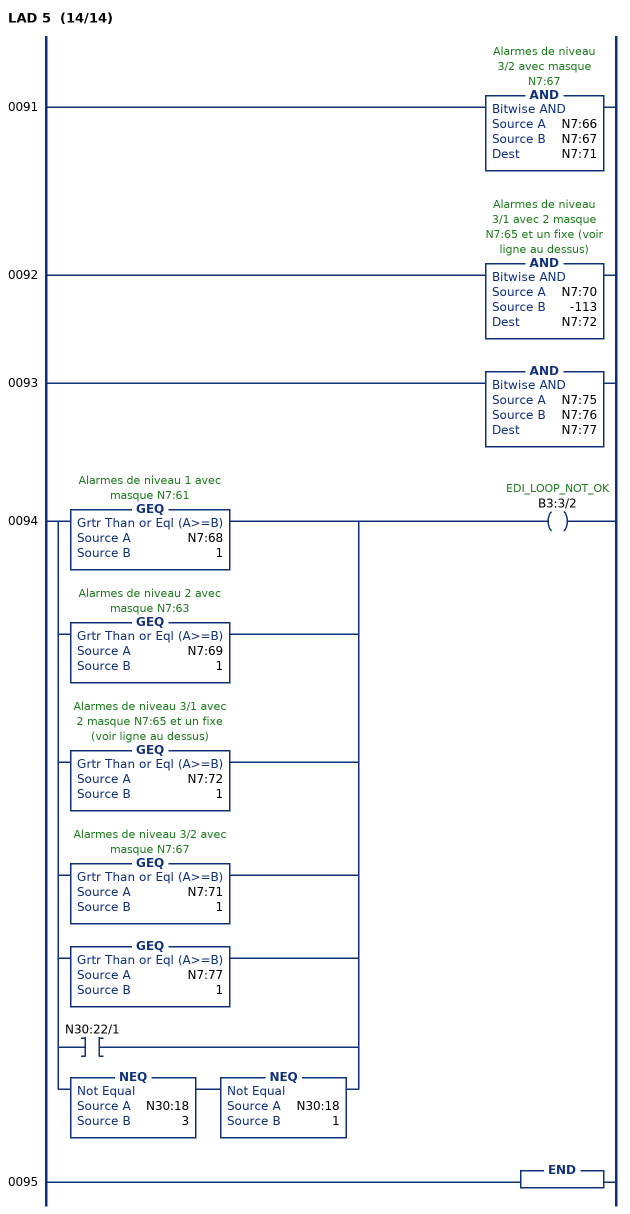
% Rung: 91 %
SOR AND N7:66 N7:67 N7:71 EOR
%   N7:71  "Alarmes de niveau 3/2 avec masque N7:67" %
% Rung: 92 %
SOR AND N7:70 -113 N7:72 EOR
%   N7:70  "Alarmes de niveau 3/1 avec masque N7:65" %
%   N7:72  "Alarmes de niveau 3/1 avec 2 masque N7:65 et un fixe (voir ligne au dessus)" %
% Rung: 93 %
SOR AND N7:75 N7:76 N7:77 EOR
% Rung: 94 %
SOR BST GEQ N7:68 1 NXB GEQ N7:69 1 NXB GEQ N7:72 1 NXB GEQ N7:71 1 NXB GEQ N7:77 1 NXB XIC N30:22/1 NXB NEQ N30:18 3 NEQ N30:18 1 BND OTE B3:3/2 EOR
%   N7:68  "Alarmes de niveau 1 avec masque N7:61" %
%   N7:69  "Alarmes de niveau 2 avec masque N7:63" %
%   N7:72  "Alarmes de niveau 3/1 avec 2 masque N7:65 et un fixe (voir ligne au dessus)" %
%   N7:71  "Alarmes de niveau 3/2 avec masque N7:67" %
%   B3:3/2  EDI_LOOP_NOT_OK %
% Rung: 95 %
SOR END EOR

LADDER 6
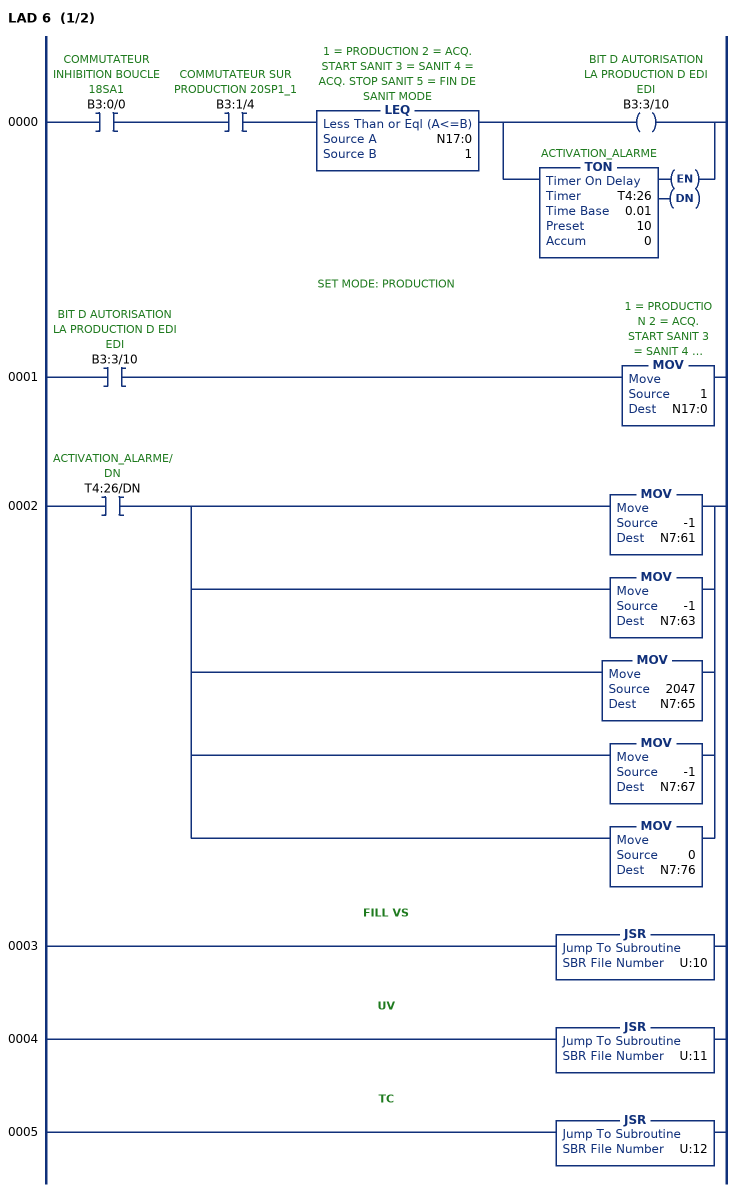
% Rung: 0 %
SOR XIC B3:0/0 XIC B3:1/4 LEQ N17:0 1 BST OTE B3:3/10 NXB TON T4:26 0.01 10 0 BND EOR
%   B3:0/0  18SA1  "COMMUTATEUR INHIBITION BOUCLE" %
%   B3:1/4  20SP1_1  "COMMUTATEUR SUR PRODUCTION" %
%   N17:0  MODE  "1 = PRODUCTION 2 = ACQ. START SANIT 3 = SANIT 4 = ACQ. STOP SANIT 5 = FIN DE SANIT" %
%   B3:3/10  EDI  "BIT D AUTORISATION LA PRODUCTION D EDI" %
%   T4:26  ACTIVATION_ALARME %
% Rung: 1 %
% SET MODE: PRODUCTION %
SOR XIC B3:3/10 MOV 1 N17:0 EOR
%   B3:3/10  EDI  "BIT D AUTORISATION LA PRODUCTION D EDI" %
%   N17:0  MODE  "1 = PRODUCTION 2 = ACQ. START SANIT 3 = SANIT 4 = ACQ. STOP SANIT 5 = FIN DE SANIT" %
% Rung: 2 %
SOR XIC T4:26/DN BST MOV -1 N7:61 NXB MOV -1 N7:63 NXB MOV 2047 N7:65 NXB MOV -1 N7:67 NXB MOV 0 N7:76 BND EOR
%   T4:26  ACTIVATION_ALARME %
% Rung: 3 %
% TITLE: FILL VS %
SOR JSR U:10 EOR
% Rung: 4 %
% TITLE: UV %
SOR JSR U:11 EOR
% Rung: 5 %
% TITLE: TC %
SOR JSR U:12 EOR

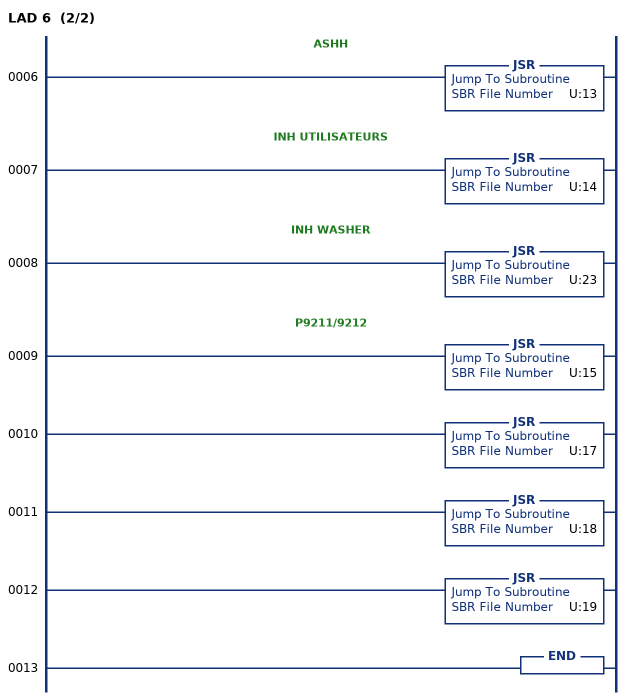
% Rung: 6 %
% TITLE: ASHH %
SOR JSR U:13 EOR
% Rung: 7 %
% TITLE: INH UTILISATEURS %
SOR JSR U:14 EOR
% Rung: 8 %
% TITLE: INH WASHER %
SOR JSR U:23 EOR
% Rung: 9 %
% TITLE: P9211/9212 %
SOR JSR U:15 EOR
% Rung: 10 %
SOR JSR U:17 EOR
% Rung: 11 %
SOR JSR U:18 EOR
% Rung: 12 %
SOR JSR U:19 EOR
% Rung: 13 %
SOR END EOR

LADDER 7
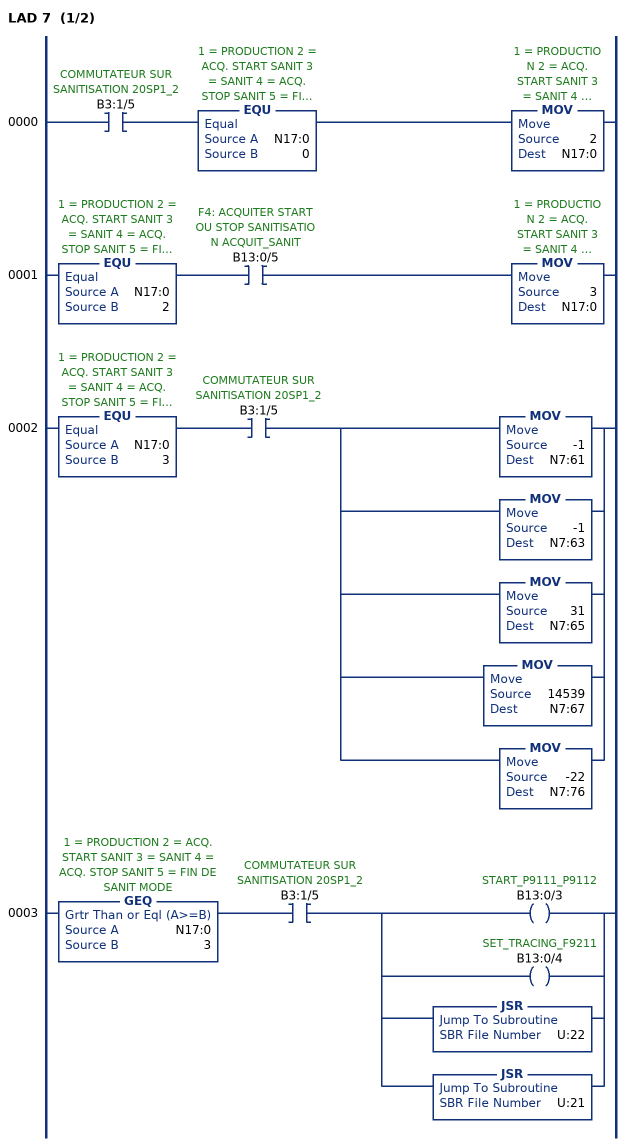
% Rung: 0 %
SOR XIC B3:1/5 EQU N17:0 0 MOV 2 N17:0 EOR
%   B3:1/5  20SP1_2  "COMMUTATEUR SUR SANITISATION" %
%   N17:0  MODE  "1 = PRODUCTION 2 = ACQ. START SANIT 3 = SANIT 4 = ACQ. STOP SANIT 5 = FIN DE SANIT" %
% Rung: 1 %
SOR EQU N17:0 2 XIC B13:0/5 MOV 3 N17:0 EOR
%   N17:0  MODE  "1 = PRODUCTION 2 = ACQ. START SANIT 3 = SANIT 4 = ACQ. STOP SANIT 5 = FIN DE SANIT" %
%   B13:0/5  ACQUIT_SANIT  "F4: ACQUITER START OU STOP SANITISATION" %
% Rung: 2 %
SOR EQU N17:0 3 XIC B3:1/5 BST MOV -1 N7:61 NXB MOV -1 N7:63 NXB MOV 31 N7:65 NXB MOV 14539 N7:67 NXB MOV -22 N7:76 BND EOR
%   N17:0  MODE  "1 = PRODUCTION 2 = ACQ. START SANIT 3 = SANIT 4 = ACQ. STOP SANIT 5 = FIN DE SANIT" %
%   B3:1/5  20SP1_2  "COMMUTATEUR SUR SANITISATION" %
% Rung: 3 %
SOR GEQ N17:0 3 XIC B3:1/5 BST OTE B13:0/3 NXB OTE B13:0/4 NXB JSR U:22 NXB JSR U:21 BND EOR
%   N17:0  MODE  "1 = PRODUCTION 2 = ACQ. START SANIT 3 = SANIT 4 = ACQ. STOP SANIT 5 = FIN DE SANIT" %
%   B3:1/5  20SP1_2  "COMMUTATEUR SUR SANITISATION" %
%   B13:0/3  START_P9111_P9112 %
%   B13:0/4  SET_TRACING_F9211 %

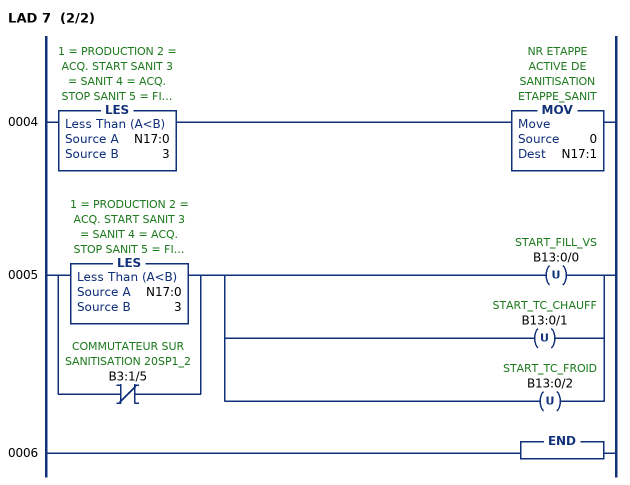
% Rung: 4 %
SOR LES N17:0 3 MOV 0 N17:1 EOR
%   N17:0  MODE  "1 = PRODUCTION 2 = ACQ. START SANIT 3 = SANIT 4 = ACQ. STOP SANIT 5 = FIN DE SANIT" %
%   N17:1  ETAPPE_SANIT  "NR ETAPPE ACTIVE DE SANITISATION" %
% Rung: 5 %
SOR BST LES N17:0 3 NXB XIO B3:1/5 BND BST OTU B13:0/0 NXB OTU B13:0/1 NXB OTU B13:0/2 BND EOR
%   N17:0  MODE  "1 = PRODUCTION 2 = ACQ. START SANIT 3 = SANIT 4 = ACQ. STOP SANIT 5 = FIN DE SANIT" %
%   B3:1/5  20SP1_2  "COMMUTATEUR SUR SANITISATION" %
%   B13:0/0  START_FILL_VS %
%   B13:0/1  START_TC_CHAUFF %
%   B13:0/2  START_TC_FROID %
% Rung: 6 %
SOR END EOR

LADDER 8
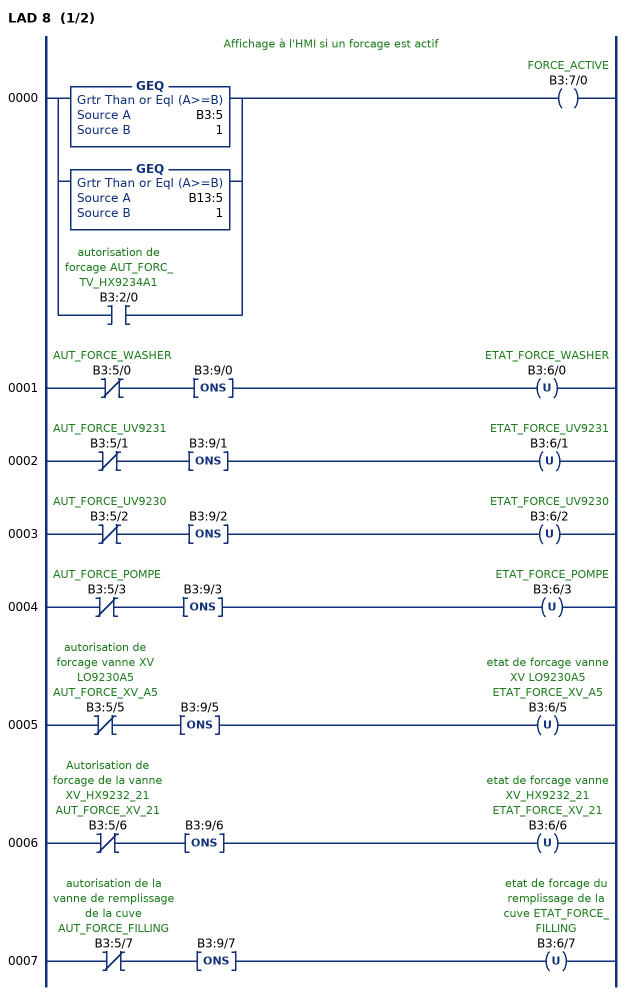
% Rung: 0 %
% Affichage à l'HMI si un forcage est actif %
SOR BST GEQ B3:5 1 NXB GEQ B13:5 1 NXB XIC B3:2/0 BND OTE B3:7/0 EOR
%   B3:2/0  AUT_FORC_TV_HX9234A1  "autorisation de forcage" %
%   B3:7/0  FORCE_ACTIVE %
% Rung: 1 %
SOR XIO B3:5/0 OSR B3:9/0 OTU B3:6/0 EOR
%   B3:5/0  AUT_FORCE_WASHER %
%   B3:6/0  ETAT_FORCE_WASHER %
% Rung: 2 %
SOR XIO B3:5/1 OSR B3:9/1 OTU B3:6/1 EOR
%   B3:5/1  AUT_FORCE_UV9231 %
%   B3:6/1  ETAT_FORCE_UV9231 %
% Rung: 3 %
SOR XIO B3:5/2 OSR B3:9/2 OTU B3:6/2 EOR
%   B3:5/2  AUT_FORCE_UV9230 %
%   B3:6/2  ETAT_FORCE_UV9230 %
% Rung: 4 %
SOR XIO B3:5/3 OSR B3:9/3 OTU B3:6/3 EOR
%   B3:5/3  AUT_FORCE_POMPE %
%   B3:6/3  ETAT_FORCE_POMPE %
% Rung: 5 %
SOR XIO B3:5/5 OSR B3:9/5 OTU B3:6/5 EOR
%   B3:5/5  AUT_FORCE_XV_A5  "autorisation de forcage vanne XV LO9230A5" %
%   B3:6/5  ETAT_FORCE_XV_A5  "etat de forcage vanne XV LO9230A5" %
% Rung: 6 %
SOR XIO B3:5/6 OSR B3:9/6 OTU B3:6/6 EOR
%   B3:5/6  AUT_FORCE_XV_21  "Autorisation de forcage de la vanne XV_HX9232_21" %
%   B3:6/6  ETAT_FORCE_XV_21  "etat de forcage vanne XV_HX9232_21" %
% Rung: 7 %
SOR XIO B3:5/7 OSR B3:9/7 OTU B3:6/7 EOR
%   B3:5/7  AUT_FORCE_FILLING  "autorisation de la vanne de remplissage de la cuve" %
%   B3:6/7  ETAT_FORCE_FILLING  "etat de forcage du remplissage de la cuve" %

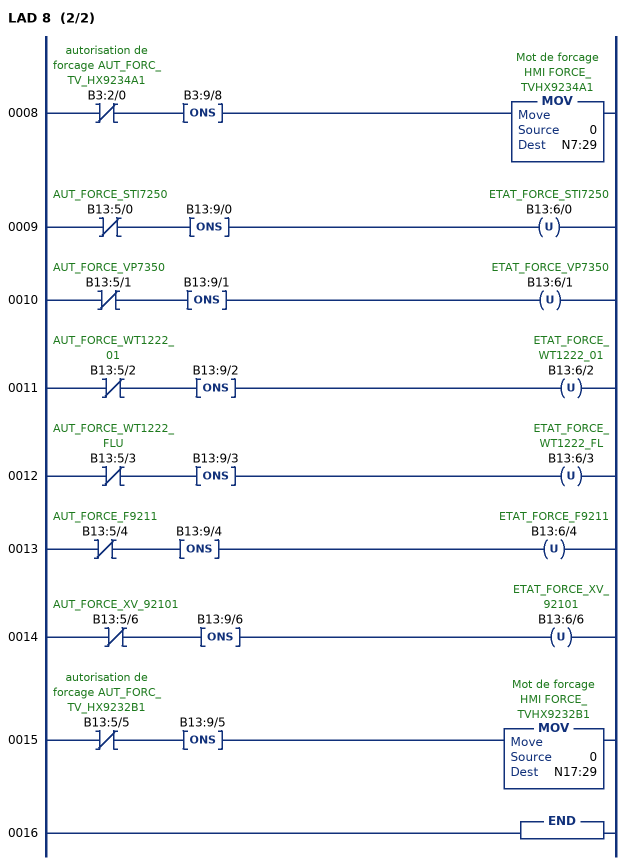
% Rung: 8 %
SOR XIO B3:2/0 OSR B3:9/8 MOV 0 N7:29 EOR
%   B3:2/0  AUT_FORC_TV_HX9234A1  "autorisation de forcage" %
%   N7:29  FORCE_TVHX9234A1  "Mot de forcage HMI" %
% Rung: 9 %
SOR XIO B13:5/0 OSR B13:9/0 OTU B13:6/0 EOR
%   B13:5/0  AUT_FORCE_STI7250 %
%   B13:6/0  ETAT_FORCE_STI7250 %
% Rung: 10 %
SOR XIO B13:5/1 OSR B13:9/1 OTU B13:6/1 EOR
%   B13:5/1  AUT_FORCE_VP7350 %
%   B13:6/1  ETAT_FORCE_VP7350 %
% Rung: 11 %
SOR XIO B13:5/2 OSR B13:9/2 OTU B13:6/2 EOR
%   B13:5/2  AUT_FORCE_WT1222_01 %
%   B13:6/2  ETAT_FORCE_WT1222_01 %
% Rung: 12 %
SOR XIO B13:5/3 OSR B13:9/3 OTU B13:6/3 EOR
%   B13:5/3  AUT_FORCE_WT1222_FLU %
%   B13:6/3  ETAT_FORCE_WT1222_FL %
% Rung: 13 %
SOR XIO B13:5/4 OSR B13:9/4 OTU B13:6/4 EOR
%   B13:5/4  AUT_FORCE_F9211 %
%   B13:6/4  ETAT_FORCE_F9211 %
% Rung: 14 %
SOR XIO B13:5/6 OSR B13:9/6 OTU B13:6/6 EOR
%   B13:5/6  "AUT_FORCE_XV_92101" %
%   B13:6/6  "ETAT_FORCE_XV_92101" %
% Rung: 15 %
SOR XIO B13:5/5 OSR B13:9/5 MOV 0 N17:29 EOR
%   B13:5/5  AUT_FORC_TV_HX9232B1  "autorisation de forcage" %
%   N17:29  FORCE_TVHX9232B1  "Mot de forcage HMI" %
% Rung: 16 %
SOR END EOR

LADDER 9
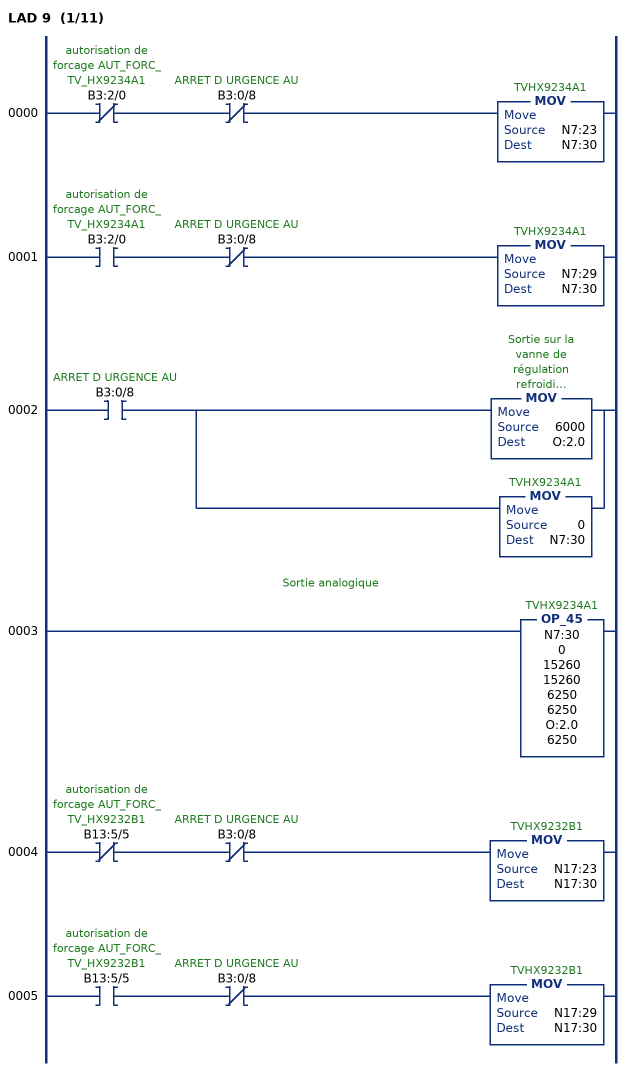
% Rung: 0 %
SOR XIO B3:2/0 XIO B3:0/8 MOV N7:23 N7:30 EOR
%   B3:2/0  AUT_FORC_TV_HX9234A1  "autorisation de forcage" %
%   B3:0/8  AU  "ARRET D URGENCE" %
%   N7:23  OUT_TC_LO9200A8  "Sortie régulateur PID" %
%   N7:30  TVHX9234A1 %
% Rung: 1 %
SOR XIC B3:2/0 XIO B3:0/8 MOV N7:29 N7:30 EOR
%   B3:2/0  AUT_FORC_TV_HX9234A1  "autorisation de forcage" %
%   B3:0/8  AU  "ARRET D URGENCE" %
%   N7:29  FORCE_TVHX9234A1  "Mot de forcage HMI" %
%   N7:30  TVHX9234A1 %
% Rung: 2 %
SOR XIC B3:0/8 BST MOV 6000 O:2.0 NXB MOV 0 N7:30 BND EOR
%   B3:0/8  AU  "ARRET D URGENCE" %
%   O:2.0  TV_HX9234A1  "Sortie sur la vanne de régulation refroidir" %
%   N7:30  TVHX9234A1 %
% Rung: 3 %
% Sortie analogique %
SOR OP_45 N7:30 0 15260 15260 6250 6250 O:2.0 6250 EOR
%   N7:30  TVHX9234A1 %
%   O:2.0  TV_HX9234A1  "Sortie sur la vanne de régulation refroidir" %
% Rung: 4 %
SOR XIO B13:5/5 XIO B3:0/8 MOV N17:23 N17:30 EOR
%   B13:5/5  AUT_FORC_TV_HX9232B1  "autorisation de forcage" %
%   B3:0/8  AU  "ARRET D URGENCE" %
%   N17:23  OUT_TC_LO9200B8  "Sortie régulateur PID" %
%   N17:30  TVHX9232B1 %
% Rung: 5 %
SOR XIC B13:5/5 XIO B3:0/8 MOV N17:29 N17:30 EOR
%   B13:5/5  AUT_FORC_TV_HX9232B1  "autorisation de forcage" %
%   B3:0/8  AU  "ARRET D URGENCE" %
%   N17:29  FORCE_TVHX9232B1  "Mot de forcage HMI" %
%   N17:30  TVHX9232B1 %

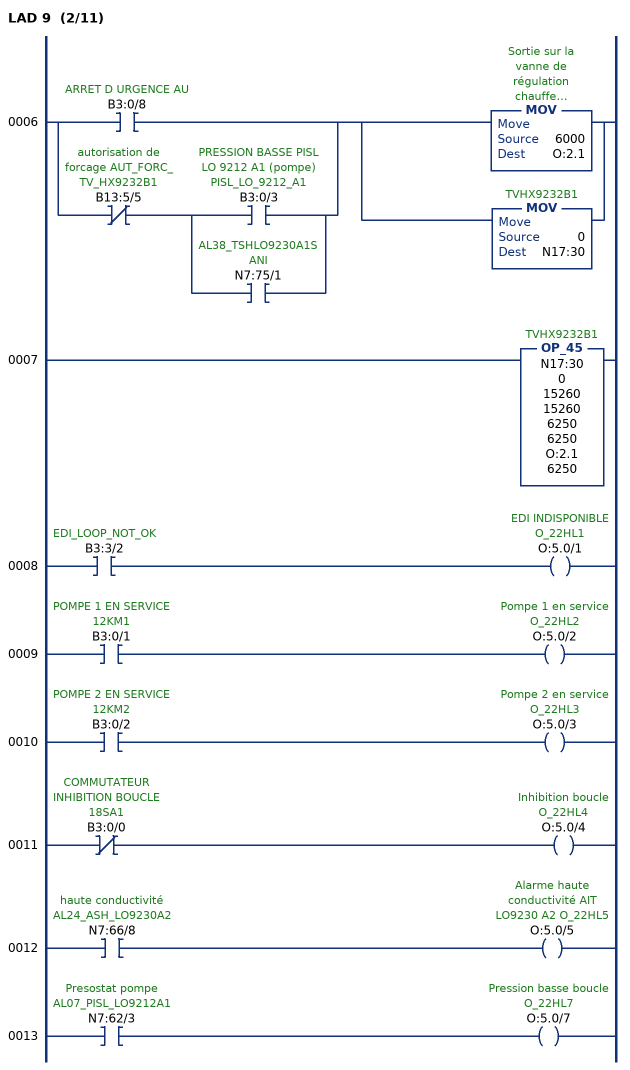
% Rung: 6 %
SOR BST XIC B3:0/8 NXB XIO B13:5/5 BST XIC B3:0/3 NXB XIC N7:75/1 BND BND BST MOV 6000 O:2.1 NXB MOV 0 N17:30 BND EOR
%   B3:0/8  AU  "ARRET D URGENCE" %
%   B13:5/5  AUT_FORC_TV_HX9232B1  "autorisation de forcage" %
%   B3:0/3  PISL_LO_9212_A1  "PRESSION BASSE PISL LO 9212 A1 (pompe)" %
%   N7:75/1  AL38_TSHLO9230A1SANI %
%   O:2.1  TV_HX9232B1  "Sortie sur la vanne de régulation chauffer" %
%   N17:30  TVHX9232B1 %
% Rung: 7 %
SOR OP_45 N17:30 0 15260 15260 6250 6250 O:2.1 6250 EOR
%   N17:30  TVHX9232B1 %
%   O:2.1  TV_HX9232B1  "Sortie sur la vanne de régulation chauffer" %
% Rung: 8 %
SOR XIC B3:3/2 OTE O:5.0/1 EOR
%   B3:3/2  EDI_LOOP_NOT_OK %
%   O:5.0/1  O_22HL1  "EDI INDISPONIBLE" %
% Rung: 9 %
SOR XIC B3:0/1 OTE O:5.0/2 EOR
%   B3:0/1  12KM1  "POMPE 1 EN SERVICE" %
%   O:5.0/2  O_22HL2  "Pompe 1 en service" %
% Rung: 10 %
SOR XIC B3:0/2 OTE O:5.0/3 EOR
%   B3:0/2  12KM2  "POMPE 2 EN SERVICE" %
%   O:5.0/3  O_22HL3  "Pompe 2 en service" %
% Rung: 11 %
SOR XIO B3:0/0 OTE O:5.0/4 EOR
%   B3:0/0  18SA1  "COMMUTATEUR INHIBITION BOUCLE" %
%   O:5.0/4  O_22HL4  "Inhibition boucle" %
% Rung: 12 %
SOR XIC N7:66/8 OTE O:5.0/5 EOR
%   N7:66/8  AL24_ASH_LO9230A2  "haute conductivité" %
%   O:5.0/5  O_22HL5  "Alarme haute conductivité AIT LO9230 A2" %
% Rung: 13 %
SOR XIC N7:62/3 OTE O:5.0/7 EOR
%   N7:62/3  AL07_PISL_LO9212A1  "Presostat pompe" %
%   O:5.0/7  O_22HL7  "Pression basse boucle" %

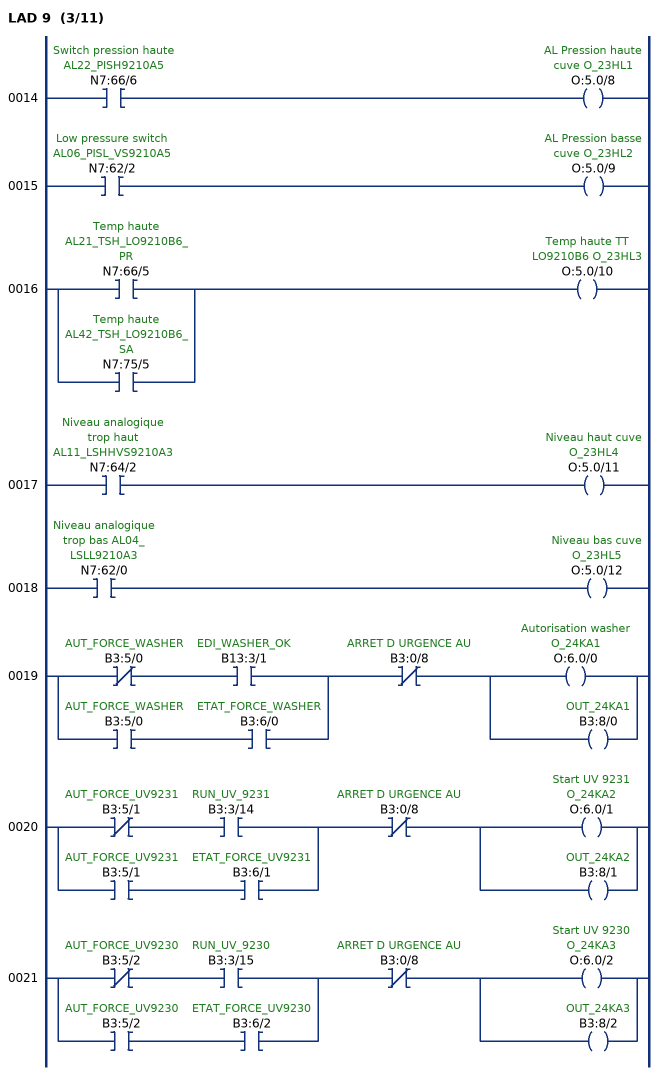
% Rung: 14 %
SOR XIC N7:66/6 OTE O:5.0/8 EOR
%   N7:66/6  AL22_PISH9210A5  "Switch pression haute" %
%   O:5.0/8  O_23HL1  "AL Pression haute cuve" %
% Rung: 15 %
SOR XIC N7:62/2 OTE O:5.0/9 EOR
%   N7:62/2  AL06_PISL_VS9210A5  "Low pressure switch" %
%   O:5.0/9  O_23HL2  "AL Pression basse cuve" %
% Rung: 16 %
SOR BST XIC N7:66/5 NXB XIC N7:75/5 BND OTE O:5.0/10 EOR
%   N7:66/5  AL21_TSH_LO9210B6_PR  "Temp haute" %
%   N7:75/5  AL42_TSH_LO9210B6_SA  "Temp haute" %
%   O:5.0/10  O_23HL3  "Temp haute TT LO9210B6" %
% Rung: 17 %
SOR XIC N7:64/2 OTE O:5.0/11 EOR
%   N7:64/2  AL11_LSHHVS9210A3  "Niveau analogique trop haut" %
%   O:5.0/11  O_23HL4  "Niveau haut cuve" %
% Rung: 18 %
SOR XIC N7:62/0 OTE O:5.0/12 EOR
%   N7:62/0  AL04_LSLL9210A3  "Niveau analogique trop bas" %
%   O:5.0/12  O_23HL5  "Niveau bas cuve" %
% Rung: 19 %
SOR BST XIO B3:5/0 XIC B13:3/1 NXB XIC B3:5/0 XIC B3:6/0 BND XIO B3:0/8 BST OTE O:6.0/0 NXB OTE B3:8/0 BND EOR
%   B3:5/0  AUT_FORCE_WASHER %
%   B13:3/1  EDI_WASHER_OK %
%   B3:6/0  ETAT_FORCE_WASHER %
%   B3:0/8  AU  "ARRET D URGENCE" %
%   O:6.0/0  O_24KA1  "Autorisation washer" %
%   B3:8/0  "OUT_24KA1" %
% Rung: 20 %
SOR BST XIO B3:5/1 XIC B3:3/14 NXB XIC B3:5/1 XIC B3:6/1 BND XIO B3:0/8 BST OTE O:6.0/1 NXB OTE B3:8/1 BND EOR
%   B3:5/1  AUT_FORCE_UV9231 %
%   B3:3/14  RUN_UV_9231 %
%   B3:6/1  ETAT_FORCE_UV9231 %
%   B3:0/8  AU  "ARRET D URGENCE" %
%   O:6.0/1  O_24KA2  "Start UV 9231" %
%   B3:8/1  "OUT_24KA2" %
% Rung: 21 %
SOR BST XIO B3:5/2 XIC B3:3/15 NXB XIC B3:5/2 XIC B3:6/2 BND XIO B3:0/8 BST OTE O:6.0/2 NXB OTE B3:8/2 BND EOR
%   B3:5/2  AUT_FORCE_UV9230 %
%   B3:3/15  RUN_UV_9230 %
%   B3:6/2  ETAT_FORCE_UV9230 %
%   B3:0/8  AU  "ARRET D URGENCE" %
%   O:6.0/2  O_24KA3  "Start UV 9230" %
%   B3:8/2  "OUT_24KA3" %

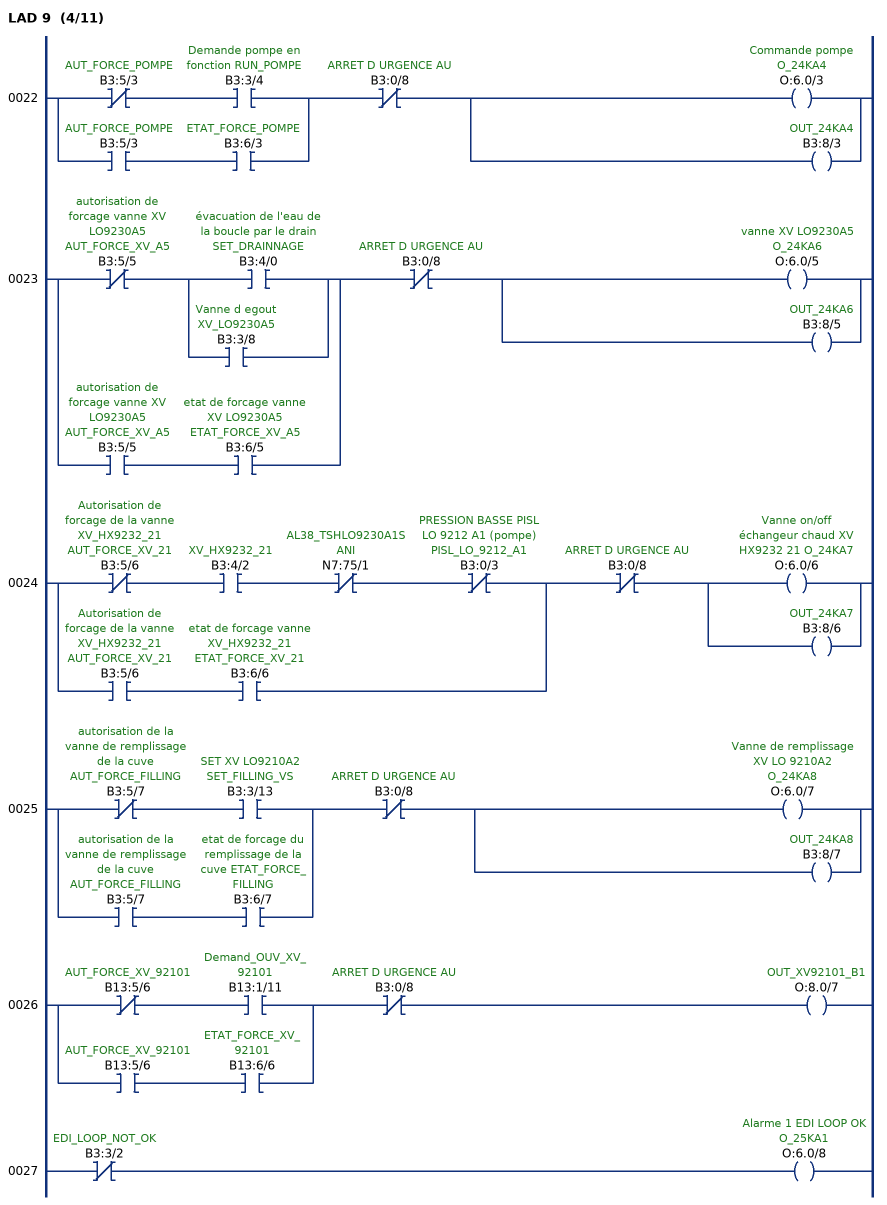
% Rung: 22 %
SOR BST XIO B3:5/3 XIC B3:3/4 NXB XIC B3:5/3 XIC B3:6/3 BND XIO B3:0/8 BST OTE O:6.0/3 NXB OTE B3:8/3 BND EOR
%   B3:5/3  AUT_FORCE_POMPE %
%   B3:3/4  RUN_POMPE  "Demande pompe en fonction" %
%   B3:6/3  ETAT_FORCE_POMPE %
%   B3:0/8  AU  "ARRET D URGENCE" %
%   O:6.0/3  O_24KA4  "Commande pompe" %
%   B3:8/3  "OUT_24KA4" %
% Rung: 23 %
SOR BST XIO B3:5/5 BST XIC B3:4/0 NXB XIC B3:3/8 BND NXB XIC B3:5/5 XIC B3:6/5 BND XIO B3:0/8 BST OTE O:6.0/5 NXB OTE B3:8/5 BND EOR
%   B3:5/5  AUT_FORCE_XV_A5  "autorisation de forcage vanne XV LO9230A5" %
%   B3:4/0  SET_DRAINNAGE  "évacuation de l'eau de la boucle par le drain" %
%   B3:3/8  XV_LO9230A5  "Vanne d egout" %
%   B3:6/5  ETAT_FORCE_XV_A5  "etat de forcage vanne XV LO9230A5" %
%   B3:0/8  AU  "ARRET D URGENCE" %
%   O:6.0/5  O_24KA6  "vanne XV LO9230A5" %
%   B3:8/5  "OUT_24KA6" %
% Rung: 24 %
SOR BST XIO B3:5/6 XIC B3:4/2 XIO N7:75/1 XIO B3:0/3 NXB XIC B3:5/6 XIC B3:6/6 BND XIO B3:0/8 BST OTE O:6.0/6 NXB OTE B3:8/6 BND EOR
%   B3:5/6  AUT_FORCE_XV_21  "Autorisation de forcage de la vanne XV_HX9232_21" %
%   B3:4/2  XV_HX9232_21 %
%   N7:75/1  AL38_TSHLO9230A1SANI %
%   B3:0/3  PISL_LO_9212_A1  "PRESSION BASSE PISL LO 9212 A1 (pompe)" %
%   B3:6/6  ETAT_FORCE_XV_21  "etat de forcage vanne XV_HX9232_21" %
%   B3:0/8  AU  "ARRET D URGENCE" %
%   O:6.0/6  O_24KA7  "Vanne on/off échangeur chaud XV HX9232 21" %
%   B3:8/6  "OUT_24KA7" %
% Rung: 25 %
SOR BST XIO B3:5/7 XIC B3:3/13 NXB XIC B3:5/7 XIC B3:6/7 BND XIO B3:0/8 BST OTE O:6.0/7 NXB OTE B3:8/7 BND EOR
%   B3:5/7  AUT_FORCE_FILLING  "autorisation de la vanne de remplissage de la cuve" %
%   B3:3/13  SET_FILLING_VS  "SET XV LO9210A2" %
%   B3:6/7  ETAT_FORCE_FILLING  "etat de forcage du remplissage de la cuve" %
%   B3:0/8  AU  "ARRET D URGENCE" %
%   O:6.0/7  O_24KA8  "Vanne de remplissage XV LO 9210A2" %
%   B3:8/7  "OUT_24KA8" %
% Rung: 26 %
SOR BST XIO B13:5/6 XIC B13:1/11 NXB XIC B13:5/6 XIC B13:6/6 BND XIO B3:0/8 OTE O:8.0/7 EOR
%   B13:5/6  "AUT_FORCE_XV_92101" %
%   B13:1/11  "Demand_OUV_XV_92101" %
%   B13:6/6  "ETAT_FORCE_XV_92101" %
%   B3:0/8  AU  "ARRET D URGENCE" %
%   O:8.0/7  "OUT_XV92101_B1" %
% Rung: 27 %
SOR XIO B3:3/2 OTE O:6.0/8 EOR
%   B3:3/2  EDI_LOOP_NOT_OK %
%   O:6.0/8  O_25KA1  "Alarme 1 EDI LOOP OK" %

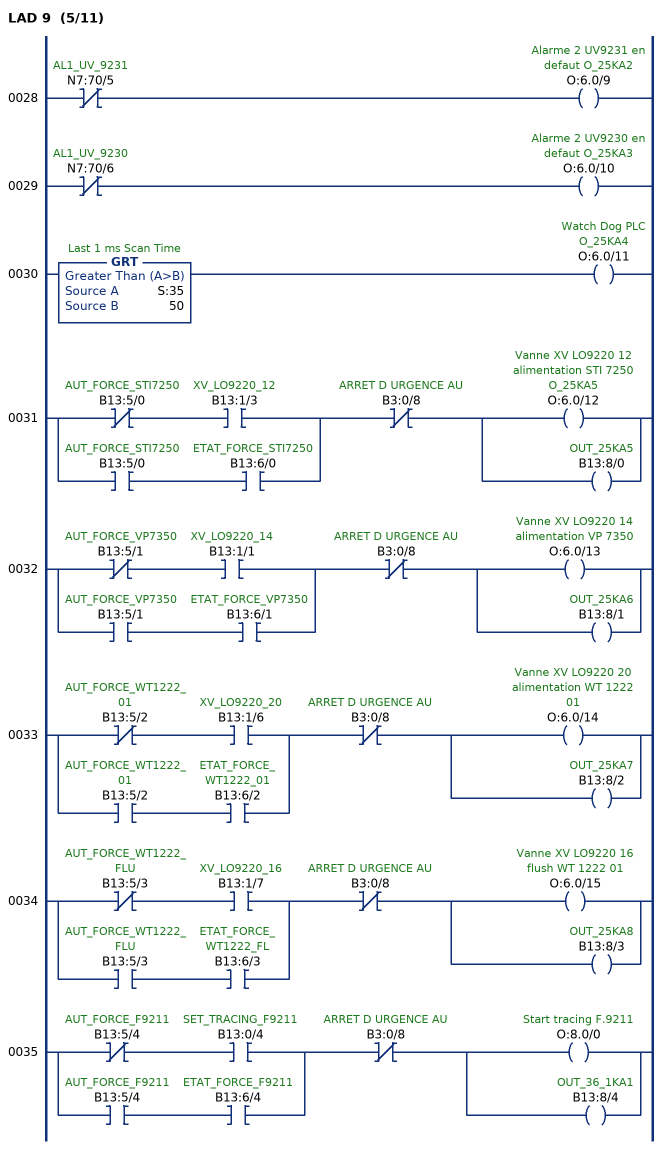
% Rung: 28 %
SOR XIO N7:70/5 OTE O:6.0/9 EOR
%   N7:70/5  AL1_UV_9231 %
%   O:6.0/9  O_25KA2  "Alarme 2 UV9231 en defaut" %
% Rung: 29 %
SOR XIO N7:70/6 OTE O:6.0/10 EOR
%   N7:70/6  AL1_UV_9230 %
%   O:6.0/10  O_25KA3  "Alarme 2 UV9230 en defaut" %
% Rung: 30 %
SOR GRT S:35 50 OTE O:6.0/11 EOR
%   S:35  "Last 1 ms Scan Time" %
%   O:6.0/11  O_25KA4  "Watch Dog PLC" %
% Rung: 31 %
SOR BST XIO B13:5/0 XIC B13:1/3 NXB XIC B13:5/0 XIC B13:6/0 BND XIO B3:0/8 BST OTE O:6.0/12 NXB OTE B13:8/0 BND EOR
%   B13:5/0  AUT_FORCE_STI7250 %
%   B13:1/3  XV_LO9220_12 %
%   B13:6/0  ETAT_FORCE_STI7250 %
%   B3:0/8  AU  "ARRET D URGENCE" %
%   O:6.0/12  O_25KA5  "Vanne XV LO9220 12 alimentation STI 7250" %
%   B13:8/0  "OUT_25KA5" %
% Rung: 32 %
SOR BST XIO B13:5/1 XIC B13:1/1 NXB XIC B13:5/1 XIC B13:6/1 BND XIO B3:0/8 BST OTE O:6.0/13 NXB OTE B13:8/1 BND EOR
%   B13:5/1  AUT_FORCE_VP7350 %
%   B13:1/1  XV_LO9220_14 %
%   B13:6/1  ETAT_FORCE_VP7350 %
%   B3:0/8  AU  "ARRET D URGENCE" %
%   O:6.0/13  "Vanne XV LO9220 14 alimentation VP 7350" %
%   B13:8/1  "OUT_25KA6" %
% Rung: 33 %
SOR BST XIO B13:5/2 XIC B13:1/6 NXB XIC B13:5/2 XIC B13:6/2 BND XIO B3:0/8 BST OTE O:6.0/14 NXB OTE B13:8/2 BND EOR
%   B13:5/2  AUT_FORCE_WT1222_01 %
%   B13:1/6  XV_LO9220_20 %
%   B13:6/2  ETAT_FORCE_WT1222_01 %
%   B3:0/8  AU  "ARRET D URGENCE" %
%   O:6.0/14  "Vanne XV LO9220 20 alimentation WT 1222 01" %
%   B13:8/2  "OUT_25KA7" %
% Rung: 34 %
SOR BST XIO B13:5/3 XIC B13:1/7 NXB XIC B13:5/3 XIC B13:6/3 BND XIO B3:0/8 BST OTE O:6.0/15 NXB OTE B13:8/3 BND EOR
%   B13:5/3  AUT_FORCE_WT1222_FLU %
%   B13:1/7  XV_LO9220_16 %
%   B13:6/3  ETAT_FORCE_WT1222_FL %
%   B3:0/8  AU  "ARRET D URGENCE" %
%   O:6.0/15  "Vanne XV LO9220 16 flush WT 1222 01" %
%   B13:8/3  "OUT_25KA8" %
% Rung: 35 %
SOR BST XIO B13:5/4 XIC B13:0/4 NXB XIC B13:5/4 XIC B13:6/4 BND XIO B3:0/8 BST OTE O:8.0/0 NXB OTE B13:8/4 BND EOR
%   B13:5/4  AUT_FORCE_F9211 %
%   B13:0/4  SET_TRACING_F9211 %
%   B13:6/4  ETAT_FORCE_F9211 %
%   B3:0/8  AU  "ARRET D URGENCE" %
%   O:8.0/0  "Start tracing F.9211" %
%   B13:8/4  "OUT_36_1KA1" %

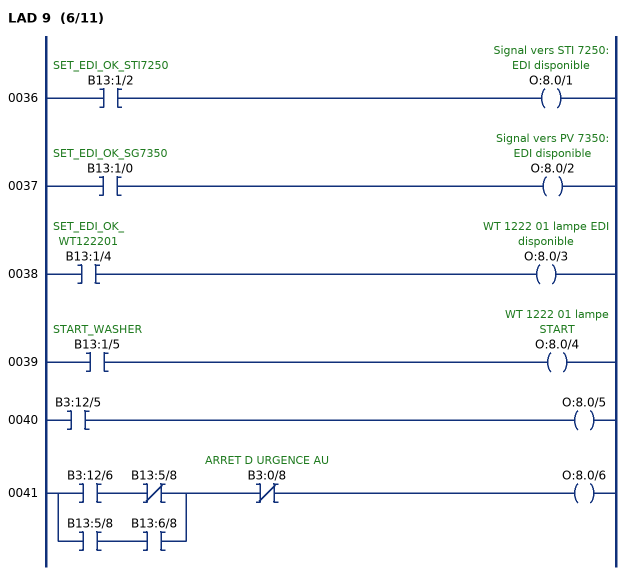
% Rung: 36 %
SOR XIC B13:1/2 OTE O:8.0/1 EOR
%   B13:1/2  SET_EDI_OK_STI7250 %
%   O:8.0/1  "Signal vers STI 7250: EDI disponible" %
% Rung: 37 %
SOR XIC B13:1/0 OTE O:8.0/2 EOR
%   B13:1/0  SET_EDI_OK_SG7350 %
%   O:8.0/2  "Signal vers PV 7350: EDI disponible" %
% Rung: 38 %
SOR XIC B13:1/4 OTE O:8.0/3 EOR
%   B13:1/4  SET_EDI_OK_WT122201 %
%   O:8.0/3  "WT 1222 01 lampe EDI disponible" %
% Rung: 39 %
SOR XIC B13:1/5 OTE O:8.0/4 EOR
%   B13:1/5  START_WASHER %
%   O:8.0/4  "WT 1222 01 lampe START" %
% Rung: 40 %
SOR XIC B3:12/5 OTE O:8.0/5 EOR
% Rung: 41 %
SOR BST XIC B3:12/6 XIO B13:5/8 NXB XIC B13:5/8 XIC B13:6/8 BND XIO B3:0/8 OTE O:8.0/6 EOR
%   B3:0/8  AU  "ARRET D URGENCE" %

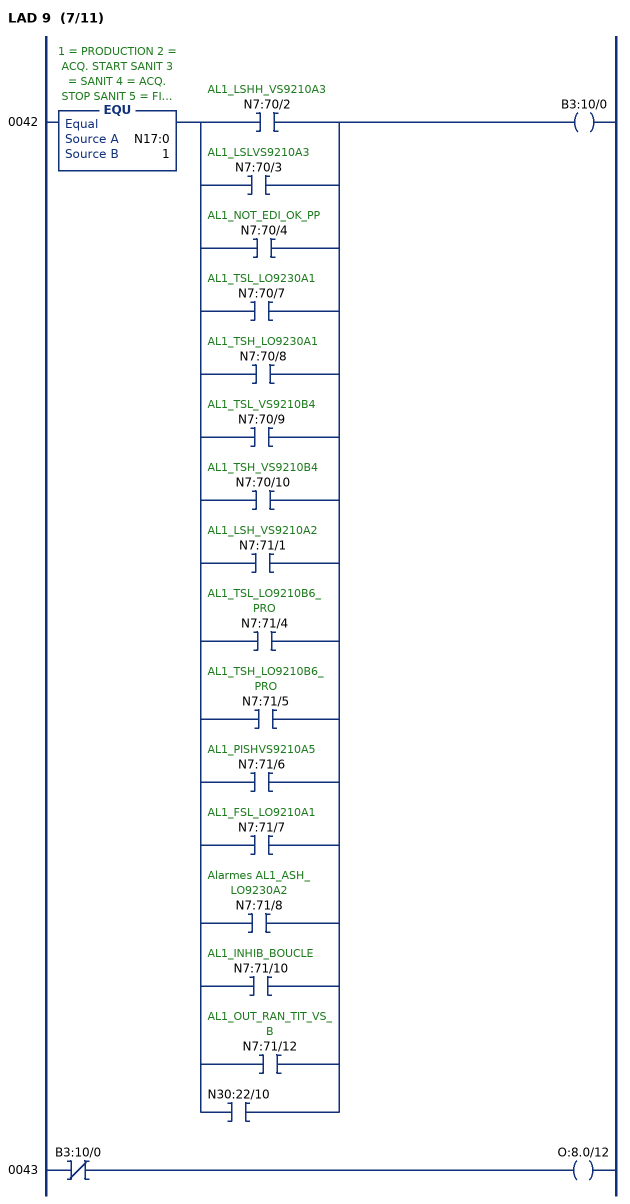
% Rung: 42 %
SOR EQU N17:0 1 BST XIC N7:70/2 NXB XIC N7:70/3 NXB XIC N7:70/4 NXB XIC N7:70/7 NXB XIC N7:70/8 NXB XIC N7:70/9 NXB XIC N7:70/10 NXB XIC N7:71/1 NXB XIC N7:71/4 NXB XIC N7:71/5 NXB XIC N7:71/6 NXB XIC N7:71/7 NXB XIC N7:71/8 NXB XIC N7:71/10 NXB XIC N7:71/12 NXB XIC N30:22/10 BND OTE B3:10/0 EOR
%   N17:0  MODE  "1 = PRODUCTION 2 = ACQ. START SANIT 3 = SANIT 4 = ACQ. STOP SANIT 5 = FIN DE SANIT" %
%   N7:70/2  AL1_LSHH_VS9210A3 %
%   N7:70/3  AL1_LSLVS9210A3 %
%   N7:70/4  AL1_NOT_EDI_OK_PP %
%   N7:70/7  AL1_TSL_LO9230A1 %
%   N7:70/8  AL1_TSH_LO9230A1 %
%   N7:70/9  AL1_TSL_VS9210B4 %
%   N7:70/10  AL1_TSH_VS9210B4 %
%   N7:71/1  AL1_LSH_VS9210A2 %
%   N7:71/4  AL1_TSL_LO9210B6_PRO %
%   N7:71/5  AL1_TSH_LO9210B6_PRO %
%   N7:71/6  AL1_PISHVS9210A5 %
%   N7:71/7  AL1_FSL_LO9210A1 %
%   N7:71/8  AL1_ASH_LO9230A2  "Alarmes" %
%   N7:71/10  AL1_INHIB_BOUCLE %
%   N7:71/12  AL1_OUT_RAN_TIT_VS_B %
% Rung: 43 %
SOR XIO B3:10/0 OTE O:8.0/12 EOR

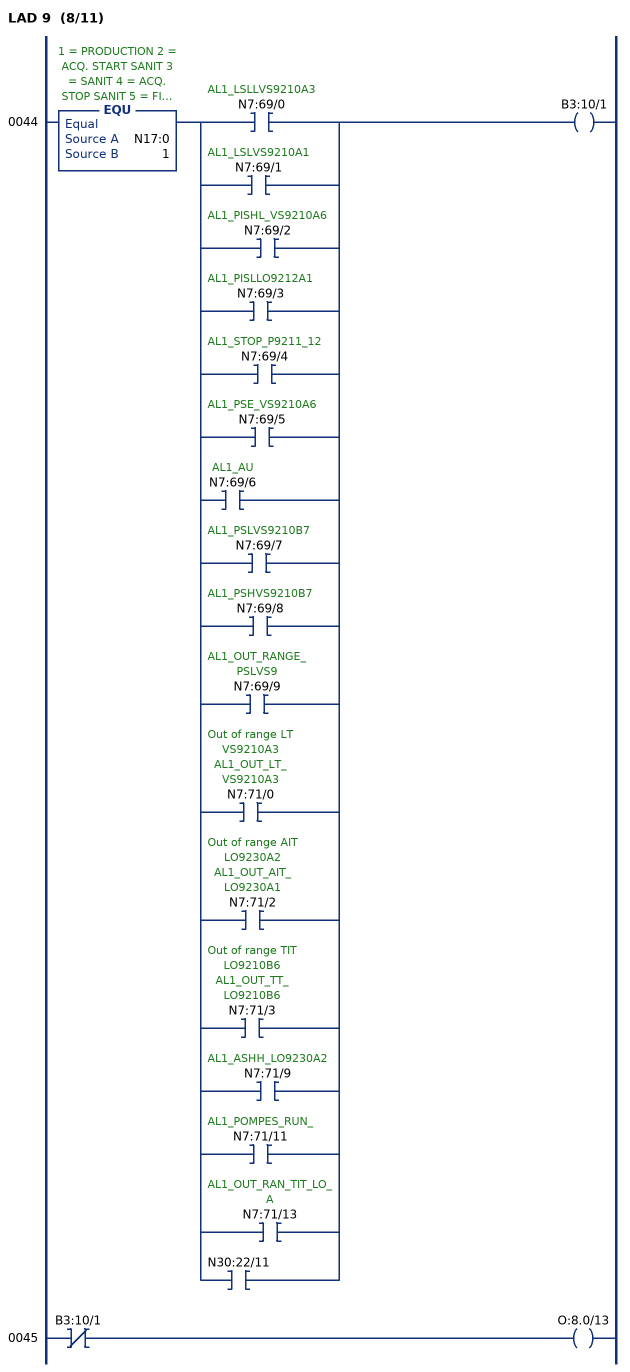
% Rung: 44 %
SOR EQU N17:0 1 BST XIC N7:69/0 NXB XIC N7:69/1 NXB XIC N7:69/2 NXB XIC N7:69/3 NXB XIC N7:69/4 NXB XIC N7:69/5 NXB XIC N7:69/6 NXB XIC N7:69/7 NXB XIC N7:69/8 NXB XIC N7:69/9 NXB XIC N7:71/0 NXB XIC N7:71/2 NXB XIC N7:71/3 NXB XIC N7:71/9 NXB XIC N7:71/11 NXB XIC N7:71/13 NXB XIC N30:22/11 BND OTE B3:10/1 EOR
%   N17:0  MODE  "1 = PRODUCTION 2 = ACQ. START SANIT 3 = SANIT 4 = ACQ. STOP SANIT 5 = FIN DE SANIT" %
%   N7:69/0  AL1_LSLLVS9210A3 %
%   N7:69/1  AL1_LSLVS9210A1 %
%   N7:69/2  AL1_PISHL_VS9210A6 %
%   N7:69/3  AL1_PISLLO9212A1 %
%   N7:69/4  AL1_STOP_P9211_12 %
%   N7:69/5  AL1_PSE_VS9210A6 %
%   N7:69/6  AL1_AU %
%   N7:69/7  AL1_PSLVS9210B7 %
%   N7:69/8  AL1_PSHVS9210B7 %
%   N7:69/9  AL1_OUT_RANGE_PSLVS9 %
%   N7:71/0  AL1_OUT_LT_VS9210A3  "Out of range LT VS9210A3" %
%   N7:71/2  AL1_OUT_AIT_LO9230A1  "Out of range AIT LO9230A2" %
%   N7:71/3  AL1_OUT_TT_LO9210B6  "Out of range TIT LO9210B6" %
%   N7:71/9  AL1_ASHH_LO9230A2 %
%   N7:71/11  AL1_POMPES_RUN_ %
%   N7:71/13  AL1_OUT_RAN_TIT_LO_A %
% Rung: 45 %
SOR XIO B3:10/1 OTE O:8.0/13 EOR

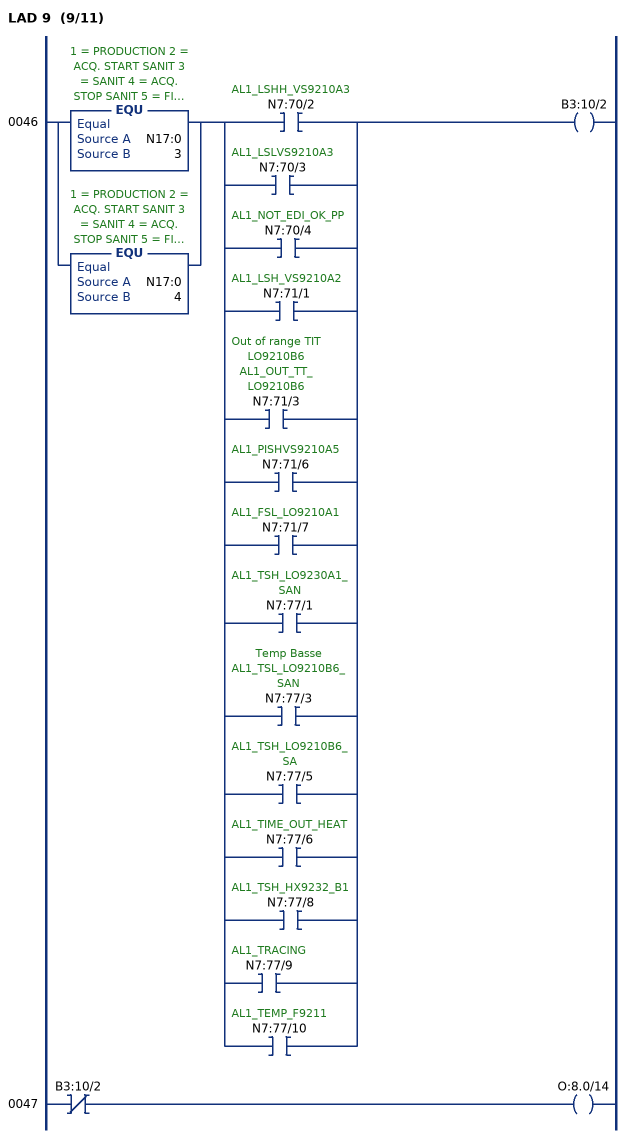
% Rung: 46 %
SOR BST EQU N17:0 3 NXB EQU N17:0 4 BND BST XIC N7:70/2 NXB XIC N7:70/3 NXB XIC N7:70/4 NXB XIC N7:71/1 NXB XIC N7:71/3 NXB XIC N7:71/6 NXB XIC N7:71/7 NXB XIC N7:77/1 NXB XIC N7:77/3 NXB XIC N7:77/5 NXB XIC N7:77/6 NXB XIC N7:77/8 NXB XIC N7:77/9 NXB XIC N7:77/10 BND OTE B3:10/2 EOR
%   N17:0  MODE  "1 = PRODUCTION 2 = ACQ. START SANIT 3 = SANIT 4 = ACQ. STOP SANIT 5 = FIN DE SANIT" %
%   N7:70/2  AL1_LSHH_VS9210A3 %
%   N7:70/3  AL1_LSLVS9210A3 %
%   N7:70/4  AL1_NOT_EDI_OK_PP %
%   N7:71/1  AL1_LSH_VS9210A2 %
%   N7:71/3  AL1_OUT_TT_LO9210B6  "Out of range TIT LO9210B6" %
%   N7:71/6  AL1_PISHVS9210A5 %
%   N7:71/7  AL1_FSL_LO9210A1 %
%   N7:77/1  AL1_TSH_LO9230A1_SAN %
%   N7:77/3  AL1_TSL_LO9210B6_SAN  "Temp Basse" %
%   N7:77/5  AL1_TSH_LO9210B6_SA %
%   N7:77/6  AL1_TIME_OUT_HEAT %
%   N7:77/8  AL1_TSH_HX9232_B1 %
%   N7:77/9  AL1_TRACING %
%   N7:77/10  AL1_TEMP_F9211 %
% Rung: 47 %
SOR XIO B3:10/2 OTE O:8.0/14 EOR

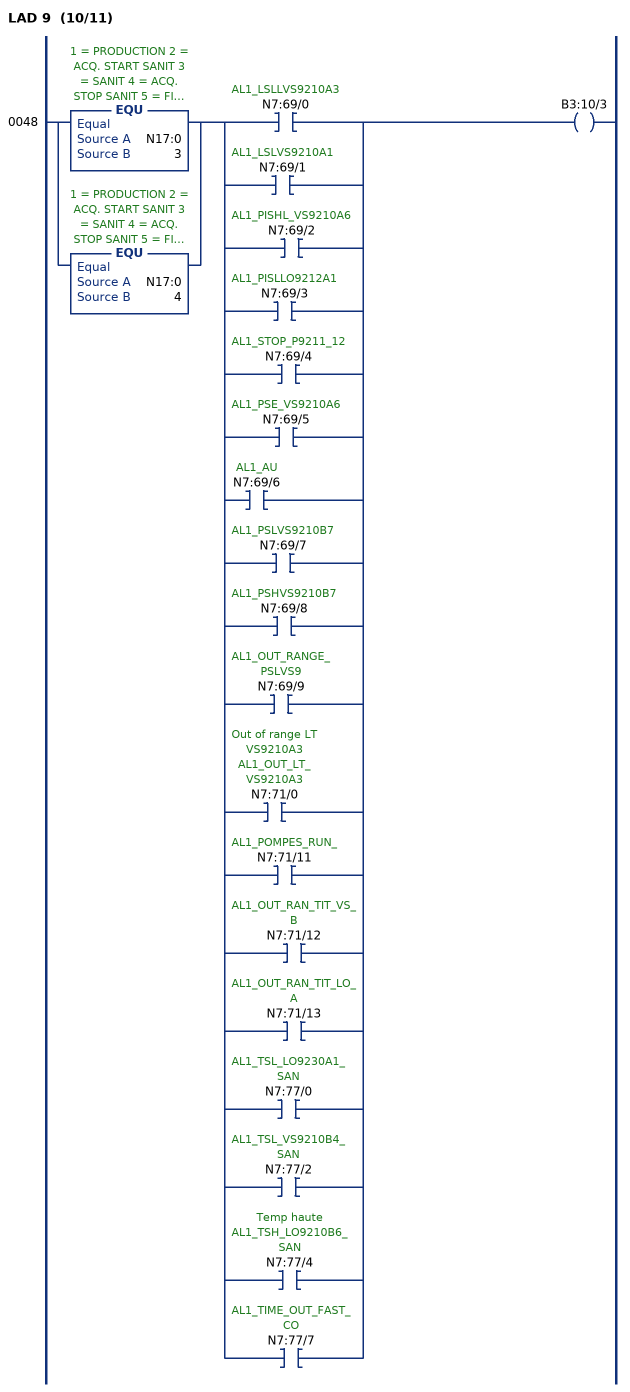
% Rung: 48 %
SOR BST EQU N17:0 3 NXB EQU N17:0 4 BND BST XIC N7:69/0 NXB XIC N7:69/1 NXB XIC N7:69/2 NXB XIC N7:69/3 NXB XIC N7:69/4 NXB XIC N7:69/5 NXB XIC N7:69/6 NXB XIC N7:69/7 NXB XIC N7:69/8 NXB XIC N7:69/9 NXB XIC N7:71/0 NXB XIC N7:71/11 NXB XIC N7:71/12 NXB XIC N7:71/13 NXB XIC N7:77/0 NXB XIC N7:77/2 NXB XIC N7:77/4 NXB XIC N7:77/7 BND OTE B3:10/3 EOR
%   N17:0  MODE  "1 = PRODUCTION 2 = ACQ. START SANIT 3 = SANIT 4 = ACQ. STOP SANIT 5 = FIN DE SANIT" %
%   N7:69/0  AL1_LSLLVS9210A3 %
%   N7:69/1  AL1_LSLVS9210A1 %
%   N7:69/2  AL1_PISHL_VS9210A6 %
%   N7:69/3  AL1_PISLLO9212A1 %
%   N7:69/4  AL1_STOP_P9211_12 %
%   N7:69/5  AL1_PSE_VS9210A6 %
%   N7:69/6  AL1_AU %
%   N7:69/7  AL1_PSLVS9210B7 %
%   N7:69/8  AL1_PSHVS9210B7 %
%   N7:69/9  AL1_OUT_RANGE_PSLVS9 %
%   N7:71/0  AL1_OUT_LT_VS9210A3  "Out of range LT VS9210A3" %
%   N7:71/11  AL1_POMPES_RUN_ %
%   N7:71/12  AL1_OUT_RAN_TIT_VS_B %
%   N7:71/13  AL1_OUT_RAN_TIT_LO_A %
%   N7:77/0  AL1_TSL_LO9230A1_SAN %
%   N7:77/2  AL1_TSL_VS9210B4_SAN %
%   N7:77/4  AL1_TSH_LO9210B6_SAN  "Temp haute" %
%   N7:77/7  AL1_TIME_OUT_FAST_CO %

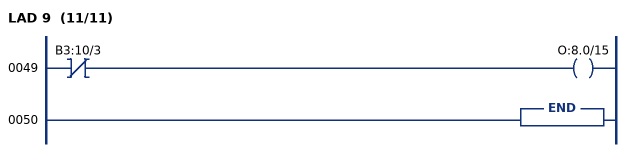
% Rung: 49 %
SOR XIO B3:10/3 OTE O:8.0/15 EOR
% Rung: 50 %
SOR END EOR

LADDER 10
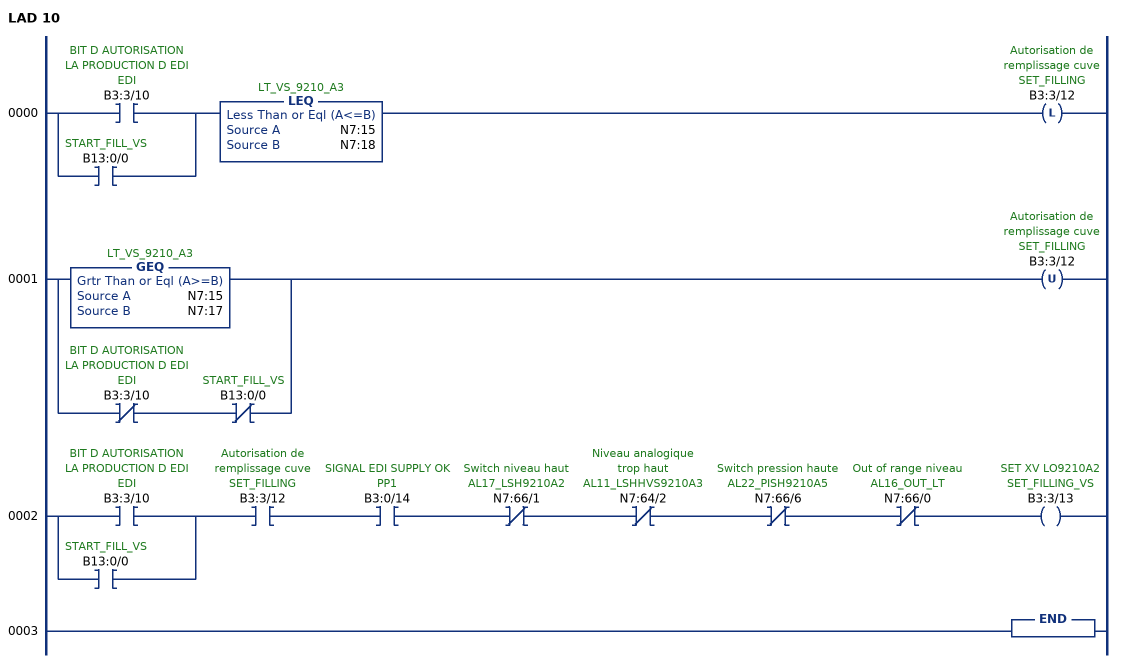
% Rung: 0 %
SOR BST XIC B3:3/10 NXB XIC B13:0/0 BND LEQ N7:15 N7:18 OTL B3:3/12 EOR
%   B3:3/10  EDI  "BIT D AUTORISATION LA PRODUCTION D EDI" %
%   B13:0/0  START_FILL_VS %
%   N7:15  LT_VS_9210_A3 %
%   N7:18  LSM_VS9210_A3_1 %
%   B3:3/12  SET_FILLING  "Autorisation de remplissage cuve" %
% Rung: 1 %
SOR BST GEQ N7:15 N7:17 NXB XIO B3:3/10 XIO B13:0/0 BND OTU B3:3/12 EOR
%   N7:15  LT_VS_9210_A3 %
%   N7:17  LSH_VS9210_A3 %
%   B3:3/10  EDI  "BIT D AUTORISATION LA PRODUCTION D EDI" %
%   B13:0/0  START_FILL_VS %
%   B3:3/12  SET_FILLING  "Autorisation de remplissage cuve" %
% Rung: 2 %
SOR BST XIC B3:3/10 NXB XIC B13:0/0 BND XIC B3:3/12 XIC B3:0/14 XIO N7:66/1 XIO N7:64/2 XIO N7:66/6 XIO N7:66/0 OTE B3:3/13 EOR
%   B3:3/10  EDI  "BIT D AUTORISATION LA PRODUCTION D EDI" %
%   B13:0/0  START_FILL_VS %
%   B3:3/12  SET_FILLING  "Autorisation de remplissage cuve" %
%   B3:0/14  PP1  "SIGNAL EDI SUPPLY OK" %
%   N7:66/1  AL17_LSH9210A2  "Switch niveau haut" %
%   N7:64/2  AL11_LSHHVS9210A3  "Niveau analogique trop haut" %
%   N7:66/6  AL22_PISH9210A5  "Switch pression haute" %
%   N7:66/0  AL16_OUT_LT  "Out of range niveau" %
%   B3:3/13  SET_FILLING_VS  "SET XV LO9210A2" %
% Rung: 3 %
SOR END EOR

LADDER 11
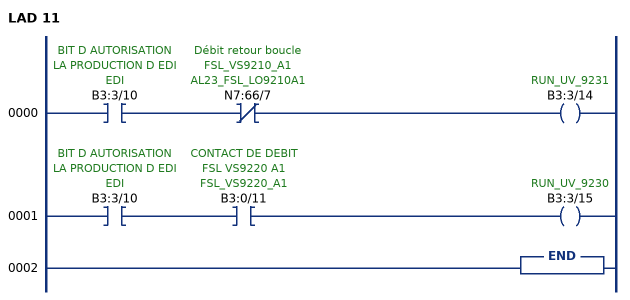
% Rung: 0 %
SOR XIC B3:3/10 XIO N7:66/7 OTE B3:3/14 EOR
%   B3:3/10  EDI  "BIT D AUTORISATION LA PRODUCTION D EDI" %
%   N7:66/7  AL23_FSL_LO9210A1  "Débit retour boucle FSL_VS9210_A1" %
%   B3:3/14  RUN_UV_9231 %
% Rung: 1 %
SOR XIC B3:3/10 XIC B3:0/11 OTE B3:3/15 EOR
%   B3:3/10  EDI  "BIT D AUTORISATION LA PRODUCTION D EDI" %
%   B3:0/11  FSL_VS9220_A1  "CONTACT DE DEBIT FSL VS9220 A1" %
%   B3:3/15  RUN_UV_9230 %
% Rung: 2 %
SOR END EOR

LADDER 12
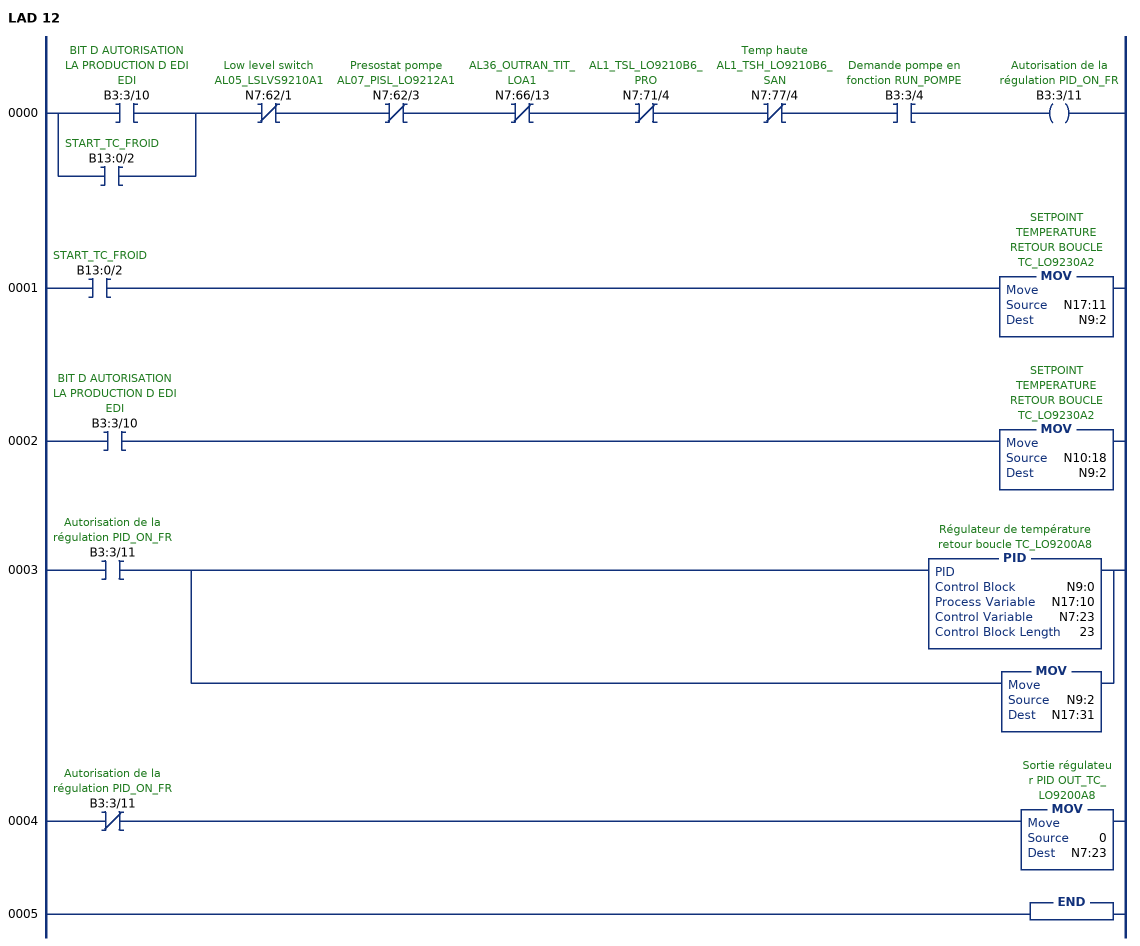
% Rung: 0 %
SOR BST XIC B3:3/10 NXB XIC B13:0/2 BND XIO N7:62/1 XIO N7:62/3 XIO N7:66/13 XIO N7:71/4 XIO N7:77/4 XIC B3:3/4 OTE B3:3/11 EOR
%   B3:3/10  EDI  "BIT D AUTORISATION LA PRODUCTION D EDI" %
%   B13:0/2  START_TC_FROID %
%   N7:62/1  AL05_LSLVS9210A1  "Low level switch" %
%   N7:62/3  AL07_PISL_LO9212A1  "Presostat pompe" %
%   N7:66/13  AL36_OUTRAN_TIT_LOA1 %
%   N7:71/4  AL1_TSL_LO9210B6_PRO %
%   N7:77/4  AL1_TSH_LO9210B6_SAN  "Temp haute" %
%   B3:3/4  RUN_POMPE  "Demande pompe en fonction" %
%   B3:3/11  PID_ON_FR  "Autorisation de la régulation" %
% Rung: 1 %
SOR XIC B13:0/2 MOV N17:11 N9:2 EOR
%   B13:0/2  START_TC_FROID %
%   N17:11  SP_COOLING %
%   N9:2  TC_LO9230A2  "SETPOINT TEMPERATURE RETOUR BOUCLE" %
% Rung: 2 %
SOR XIC B3:3/10 MOV N10:18 N9:2 EOR
%   B3:3/10  EDI  "BIT D AUTORISATION LA PRODUCTION D EDI" %
%   N10:18  SP_TEMP_PROD %
%   N9:2  TC_LO9230A2  "SETPOINT TEMPERATURE RETOUR BOUCLE" %
% Rung: 3 %
SOR XIC B3:3/11 BST PID N9:0 N17:10 N7:23 23 NXB MOV N9:2 N17:31 BND EOR
%   B3:3/11  PID_ON_FR  "Autorisation de la régulation" %
%   N9:0  TC_LO9200A8  "Régulateur de température retour boucle" %
%   N17:10  TIT_LO9230_A1 %
%   N7:23  OUT_TC_LO9200A8  "Sortie régulateur PID" %
%   N9:2  TC_LO9230A2  "SETPOINT TEMPERATURE RETOUR BOUCLE" %
% Rung: 4 %
SOR XIO B3:3/11 MOV 0 N7:23 EOR
%   B3:3/11  PID_ON_FR  "Autorisation de la régulation" %
%   N7:23  OUT_TC_LO9200A8  "Sortie régulateur PID" %
% Rung: 5 %
SOR END EOR

LADDER 13
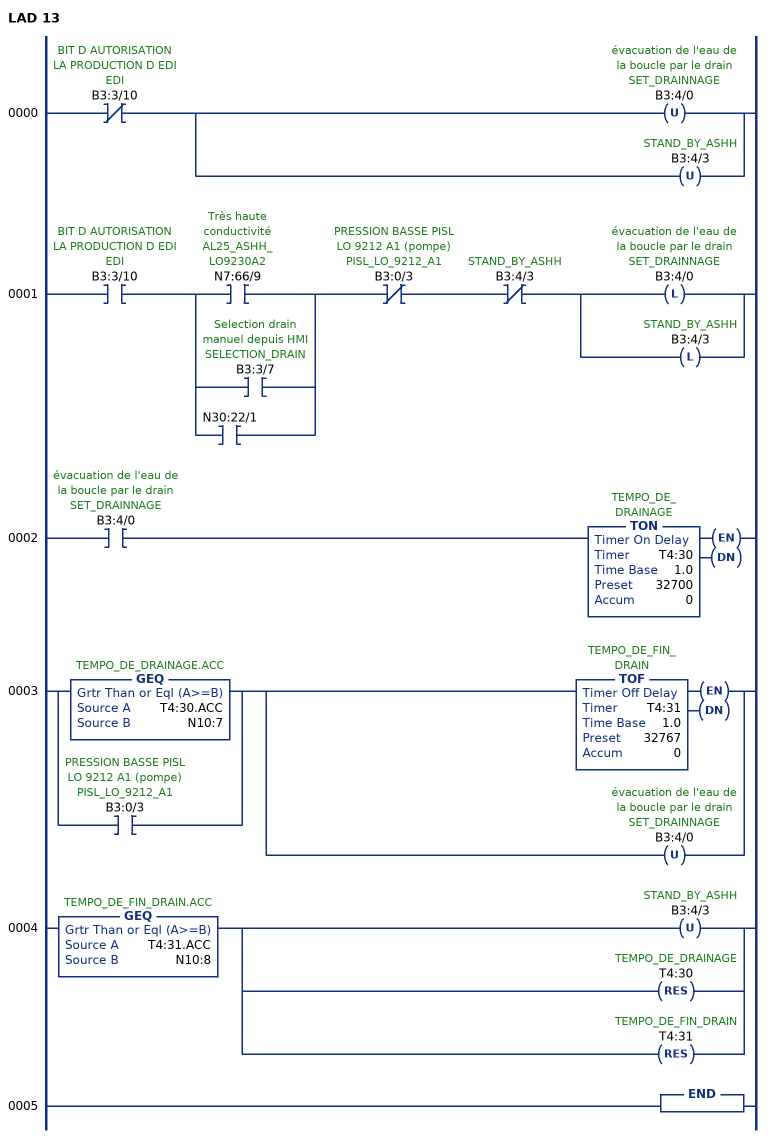
% Rung: 0 %
SOR XIO B3:3/10 BST OTU B3:4/0 NXB OTU B3:4/3 BND EOR
%   B3:3/10  EDI  "BIT D AUTORISATION LA PRODUCTION D EDI" %
%   B3:4/0  SET_DRAINNAGE  "évacuation de l'eau de la boucle par le drain" %
%   B3:4/3  STAND_BY_ASHH %
% Rung: 1 %
SOR XIC B3:3/10 BST XIC N7:66/9 NXB XIC B3:3/7 NXB XIC N30:22/1 BND XIO B3:0/3 XIO B3:4/3 BST OTL B3:4/0 NXB OTL B3:4/3 BND EOR
%   B3:3/10  EDI  "BIT D AUTORISATION LA PRODUCTION D EDI" %
%   N7:66/9  AL25_ASHH_LO9230A2  "Très haute conductivité" %
%   B3:3/7  SELECTION_DRAIN  "Selection drain manuel depuis HMI" %
%   B3:0/3  PISL_LO_9212_A1  "PRESSION BASSE PISL LO 9212 A1 (pompe)" %
%   B3:4/3  STAND_BY_ASHH %
%   B3:4/0  SET_DRAINNAGE  "évacuation de l'eau de la boucle par le drain" %
% Rung: 2 %
SOR XIC B3:4/0 TON T4:30 1.0 32700 0 EOR
%   B3:4/0  SET_DRAINNAGE  "évacuation de l'eau de la boucle par le drain" %
%   T4:30  TEMPO_DE_DRAINAGE %
% Rung: 3 %
SOR BST GEQ T4:30.ACC N10:7 NXB XIC B3:0/3 BND BST TOF T4:31 1.0 32767 0 NXB OTU B3:4/0 BND EOR
%   T4:30  TEMPO_DE_DRAINAGE %
%   N10:7  TPS_DRAINNAGE %
%   B3:0/3  PISL_LO_9212_A1  "PRESSION BASSE PISL LO 9212 A1 (pompe)" %
%   T4:31  TEMPO_DE_FIN_DRAIN %
%   B3:4/0  SET_DRAINNAGE  "évacuation de l'eau de la boucle par le drain" %
% Rung: 4 %
SOR GEQ T4:31.ACC N10:8 BST OTU B3:4/3 NXB RES T4:30 NXB RES T4:31 BND EOR
%   T4:31  TEMPO_DE_FIN_DRAIN %
%   N10:8  TPS_PAUSE_DRAINNAGE %
%   B3:4/3  STAND_BY_ASHH %
%   T4:30  TEMPO_DE_DRAINAGE %
% Rung: 5 %
SOR END EOR

LADDER 14
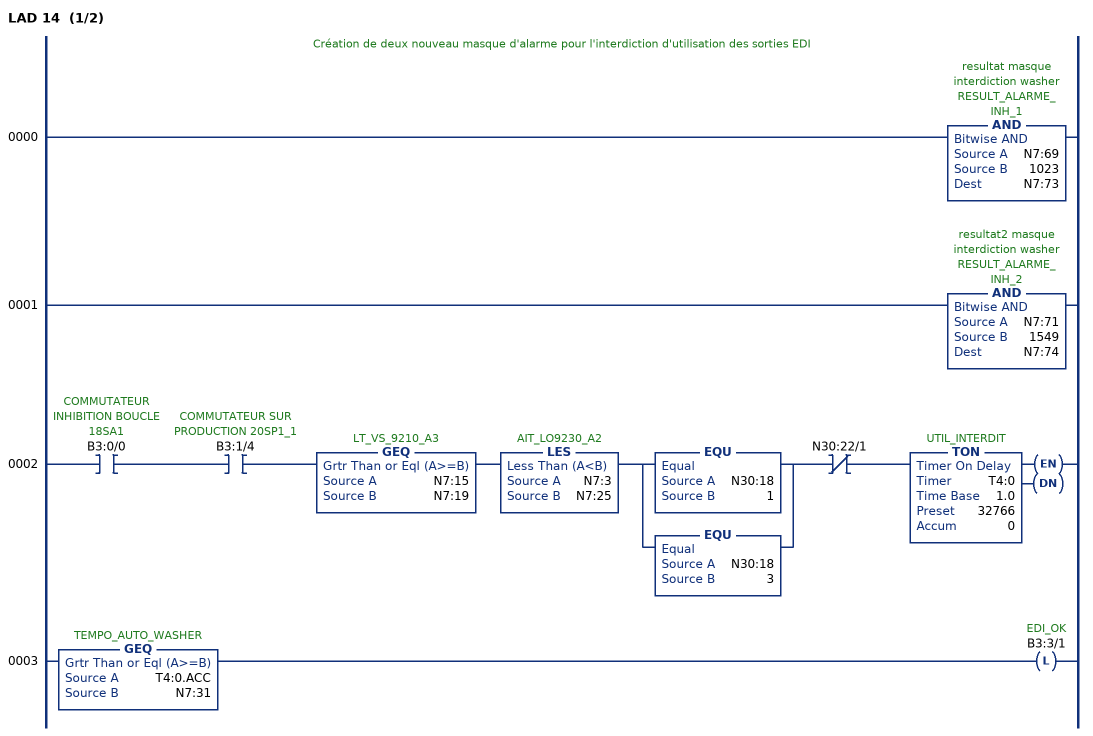
% Rung: 0 %
% Création de deux nouveau masque d'alarme pour l'interdiction d'utilisation des sorties EDI %
SOR AND N7:69 1023 N7:73 EOR
%   N7:69  "Alarmes de niveau 2 avec masque N7:63" %
%   N7:73  RESULT_ALARME_INH_1  "resultat masque interdiction washer" %
% Rung: 1 %
SOR AND N7:71 1549 N7:74 EOR
%   N7:71  "Alarmes de niveau 3/2 avec masque N7:67" %
%   N7:74  RESULT_ALARME_INH_2  "resultat2 masque interdiction washer" %
% Rung: 2 %
SOR XIC B3:0/0 XIC B3:1/4 GEQ N7:15 N7:19 LES N7:3 N7:25 BST EQU N30:18 1 NXB EQU N30:18 3 BND XIO N30:22/1 TON T4:0 1.0 32766 0 EOR
%   B3:0/0  18SA1  "COMMUTATEUR INHIBITION BOUCLE" %
%   B3:1/4  20SP1_1  "COMMUTATEUR SUR PRODUCTION" %
%   N7:15  LT_VS_9210_A3 %
%   N7:19  LSM_VS9210_A3_2 %
%   N7:3  AIT_LO9230_A2 %
%   N7:25  ASHH_LO9230A2  "HIGH HIGH CONDUCTIVITE RETURN" %
%   T4:0  UTIL_INTERDIT %
% Rung: 3 %
SOR GEQ T4:0.ACC N7:31 OTL B3:3/1 EOR
%   T4:0.ACC  TEMPO_AUTO_WASHER %
%   N7:31  TEMPO_WASHER %
%   B3:3/1  EDI_OK %

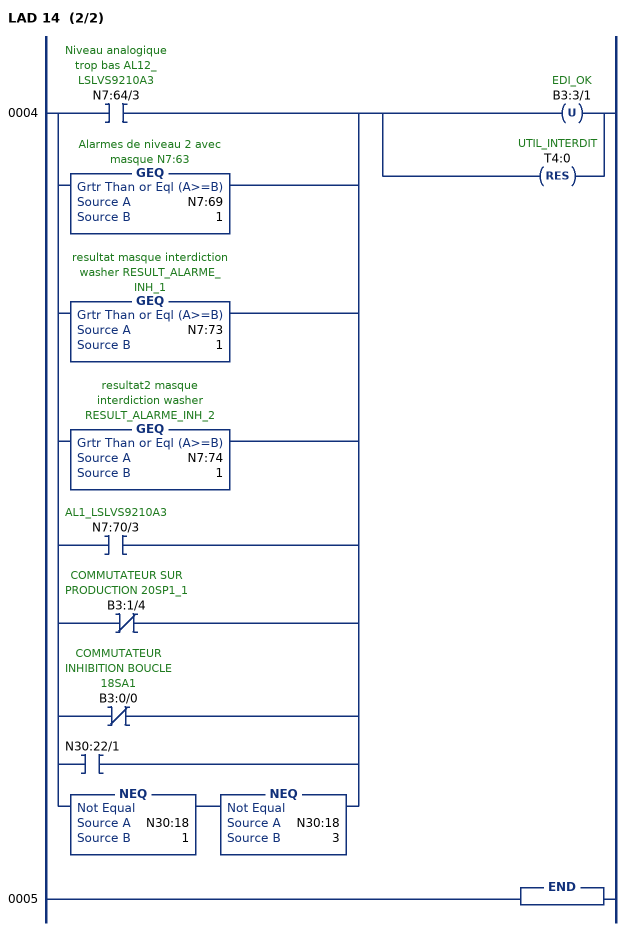
% Rung: 4 %
SOR BST XIC N7:64/3 NXB GEQ N7:69 1 NXB GEQ N7:73 1 NXB GEQ N7:74 1 NXB XIC N7:70/3 NXB XIO B3:1/4 NXB XIO B3:0/0 NXB XIC N30:22/1 NXB NEQ N30:18 1 NEQ N30:18 3 BND BST OTU B3:3/1 NXB RES T4:0 BND EOR
%   N7:64/3  AL12_LSLVS9210A3  "Niveau analogique trop bas" %
%   N7:69  "Alarmes de niveau 2 avec masque N7:63" %
%   N7:73  RESULT_ALARME_INH_1  "resultat masque interdiction washer" %
%   N7:74  RESULT_ALARME_INH_2  "resultat2 masque interdiction washer" %
%   N7:70/3  AL1_LSLVS9210A3 %
%   B3:1/4  20SP1_1  "COMMUTATEUR SUR PRODUCTION" %
%   B3:0/0  18SA1  "COMMUTATEUR INHIBITION BOUCLE" %
%   B3:3/1  EDI_OK %
%   T4:0  UTIL_INTERDIT %
% Rung: 5 %
SOR END EOR

LADDER 15
